FUNCTION_BLOCK EL2712
VAR
	{attribute addProperty Name "WcState"}
	_wcState : WcStateBase;
	{attribute addProperty Name "Info data"}
	_infoData : InfoDataBase;
	_io : EL2xx2_Data;
END_VAR

PROPERTY IO : REFERENCE TO EL2xx2_Data
GET
IO REF= _io;
END_GET
END_PROPERTY

PROPERTY WcState : REFERENCE TO WcStateBase
GET
WcState REF= _wcState;
END_GET
END_PROPERTY

END_FUNCTION_BLOCK

(* stored: Version 1.1.0.1, ProductVersion 3.1.4024.9
   POU EL2712: Id {d5209774-0c46-0cb3-09ed-ef307dfb0bf0}, SpecialFunc None
   Property IO: Id {757ce4ff-b00b-01c7-2762-fb1bc9058f79}
   Get Get: Id {bb2fa509-e493-0a76-3437-2b8df2489c1b}
   Property WcState: Id {ae97ac85-02f1-0800-2389-0a050daa27c0}
   Get Get: Id {23ad4620-939d-070b-2ca2-d4c1999eae07} *)
